(* Logix 5000 project; controller R5_CSS vendor 1 type 14 code 74 rev 19.11; software revision 19.01; part 11 of 18 *)
(* tags used below, declared in another part *)
   P205 : PUMP_CONTROL;   // OVERHEAD CONDENSER TRANSFER PUMP
   PC101 : PRESSURE_CONTROL;   // Upper quench tower Diff Pressure
   PC101A : PRESSURE_CONTROL;   // LOWER QUENCH TOWER PRESSURE TRANSMITTER
   PC101B : PRESSURE_CONTROL;   // UPPER QUENCH TOWER PRESSURE TRANSMITTER PRESSURE CONTOL
   PC102A : PRESSURE_CONTROL;   // QUENCH BASIN TRANSFER PUMP SUCTION PRESSURE CONTROL
   PC102B : PRESSURE_CONTROL;   // QUENCH BASIN TRANSFER PUMP DISCHARGE PRESSURE CONTROL
   PC132 : PRESSURE_CONTROL;
   PC132_AUTO_Ons : BOOL;
   PC132_AUTO_Ons1 : BOOL;
   PC132_PID : PID;
   PC132_PID_TON : TIMER;
   PC133 : PRESSURE_CONTROL;
   PC133_AUTO_Ons : BOOL;
   PC133_AUTO_Ons1 : BOOL;
   PC133_PID : PID;
   PC133_PID_TON : TIMER;
   Test : INT[500];
   TMR_CRIT_FAULT : DINT;
   TMR_FAULT : DINT;
(* MainProgram, continued *)

ROUTINE PC101_QuenchTowerPressureDelta   (* ladder *)
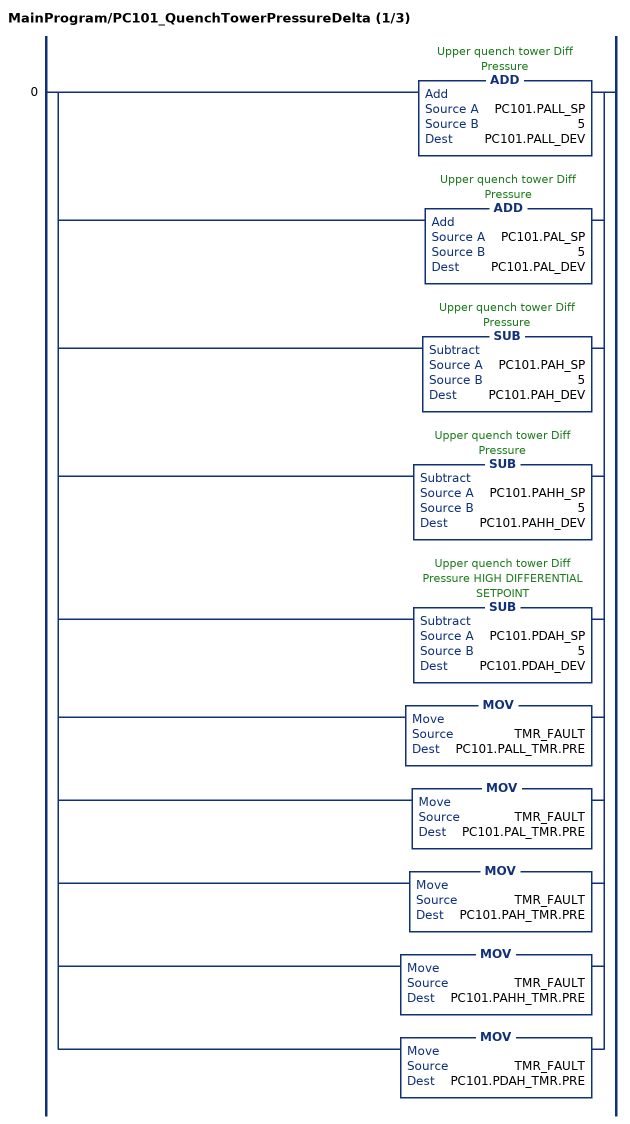
   0: [ADD(PC101.PALL_SP,5,PC101.PALL_DEV) ,ADD(PC101.PAL_SP,5,PC101.PAL_DEV) ,SUB(PC101.PAH_SP,5,PC101.PAH_DEV) ,SUB(PC101.PAHH_SP,5,PC101.PAHH_DEV) ,SUB(PC101.PDAH_SP,5,PC101.PDAH_DEV) ,MOV(TMR_FAULT,PC101.PALL_TMR.PRE) ,MOV(TMR_FAULT,PC101.PAL_TMR.PRE) ,MOV(TMR_FAULT,PC101.PAH_TMR.PRE) ,MOV(TMR_FAULT,PC101.PAHH_TMR.PRE) ,MOV(TMR_FAULT,PC101.PDAH_TMR.PRE) ];
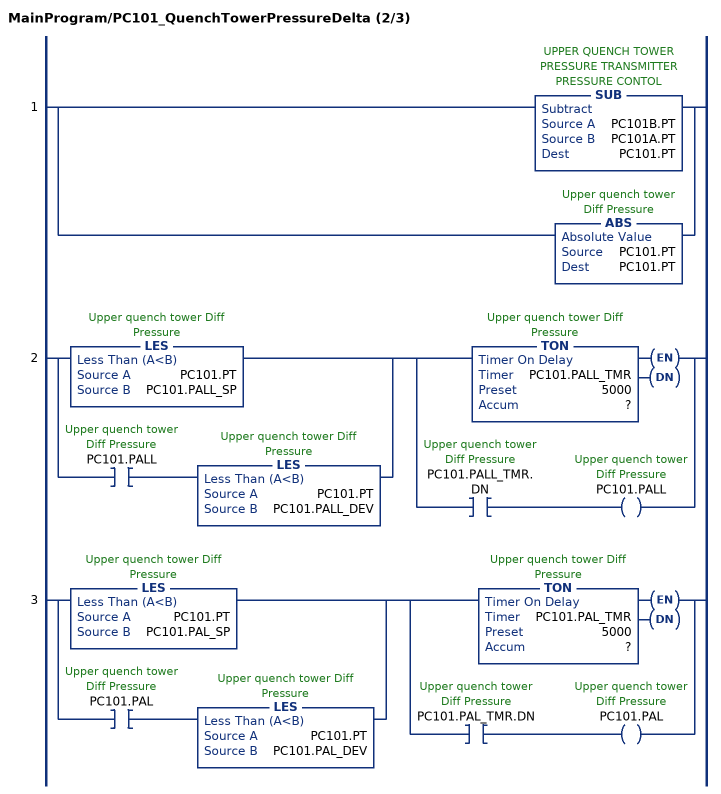
   1: [SUB(PC101B.PT,PC101A.PT,PC101.PT) ,ABS(PC101.PT,PC101.PT) ];
   2: [LES(PC101.PT,PC101.PALL_SP) ,XIC(PC101.PALL) LES(PC101.PT,PC101.PALL_DEV) ][TON(PC101.PALL_TMR,?,?) ,XIC(PC101.PALL_TMR.DN) OTE(PC101.PALL) ];
   3: [LES(PC101.PT,PC101.PAL_SP) ,XIC(PC101.PAL) LES(PC101.PT,PC101.PAL_DEV) ][TON(PC101.PAL_TMR,?,?) ,XIC(PC101.PAL_TMR.DN) OTE(PC101.PAL) ];
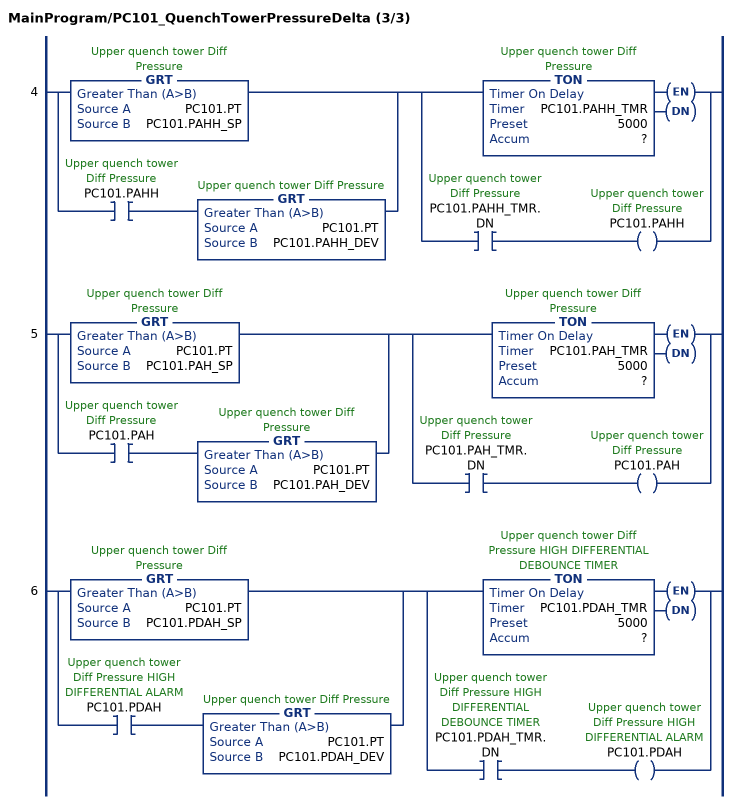
   4: [GRT(PC101.PT,PC101.PAHH_SP) ,XIC(PC101.PAHH) GRT(PC101.PT,PC101.PAHH_DEV) ][TON(PC101.PAHH_TMR,?,?) ,XIC(PC101.PAHH_TMR.DN) OTE(PC101.PAHH) ];
   5: [GRT(PC101.PT,PC101.PAH_SP) ,XIC(PC101.PAH) GRT(PC101.PT,PC101.PAH_DEV) ][TON(PC101.PAH_TMR,?,?) ,XIC(PC101.PAH_TMR.DN) OTE(PC101.PAH) ];
   6: [GRT(PC101.PT,PC101.PDAH_SP) ,XIC(PC101.PDAH) GRT(PC101.PT,PC101.PDAH_DEV) ][TON(PC101.PDAH_TMR,?,?) ,XIC(PC101.PDAH_TMR.DN) OTE(PC101.PDAH) ];
END_ROUTINE

ROUTINE PC101A_QuenchTowerPressure   (* ladder *)
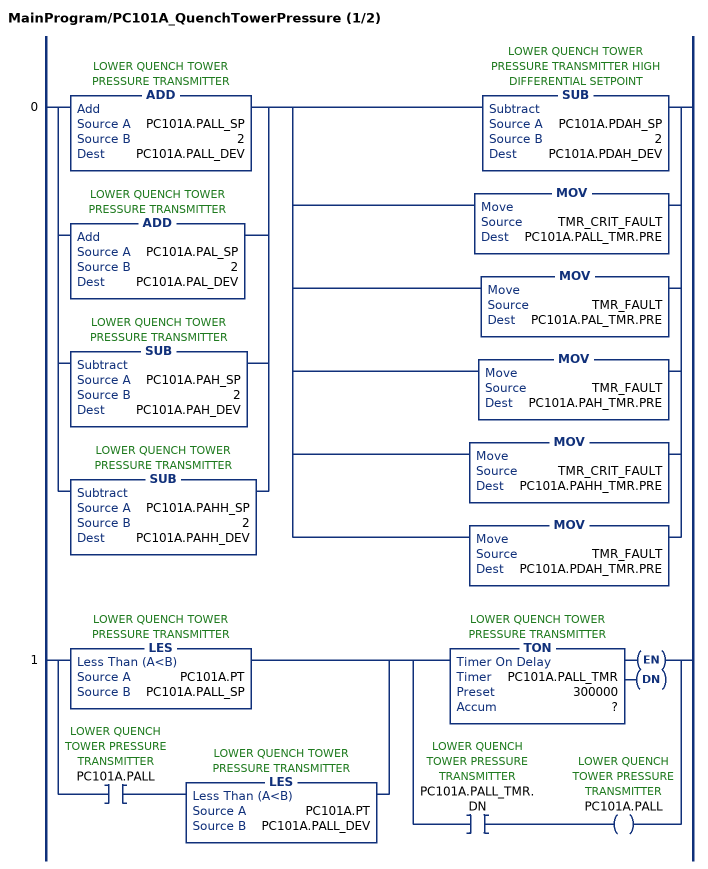
   0: [ADD(PC101A.PALL_SP,2,PC101A.PALL_DEV) ,ADD(PC101A.PAL_SP,2,PC101A.PAL_DEV) ,SUB(PC101A.PAH_SP,2,PC101A.PAH_DEV) ,SUB(PC101A.PAHH_SP,2,PC101A.PAHH_DEV) ][SUB(PC101A.PDAH_SP,2,PC101A.PDAH_DEV) ,MOV(TMR_CRIT_FAULT,PC101A.PALL_TMR.PRE) ,MOV(TMR_FAULT,PC101A.PAL_TMR.PRE) ,MOV(TMR_FAULT,PC101A.PAH_TMR.PRE) ,MOV(TMR_CRIT_FAULT,PC101A.PAHH_TMR.PRE) ,MOV(TMR_FAULT,PC101A.PDAH_TMR.PRE) ];
   1: [LES(PC101A.PT,PC101A.PALL_SP) ,XIC(PC101A.PALL) LES(PC101A.PT,PC101A.PALL_DEV) ][TON(PC101A.PALL_TMR,?,?) ,XIC(PC101A.PALL_TMR.DN) OTE(PC101A.PALL) ];
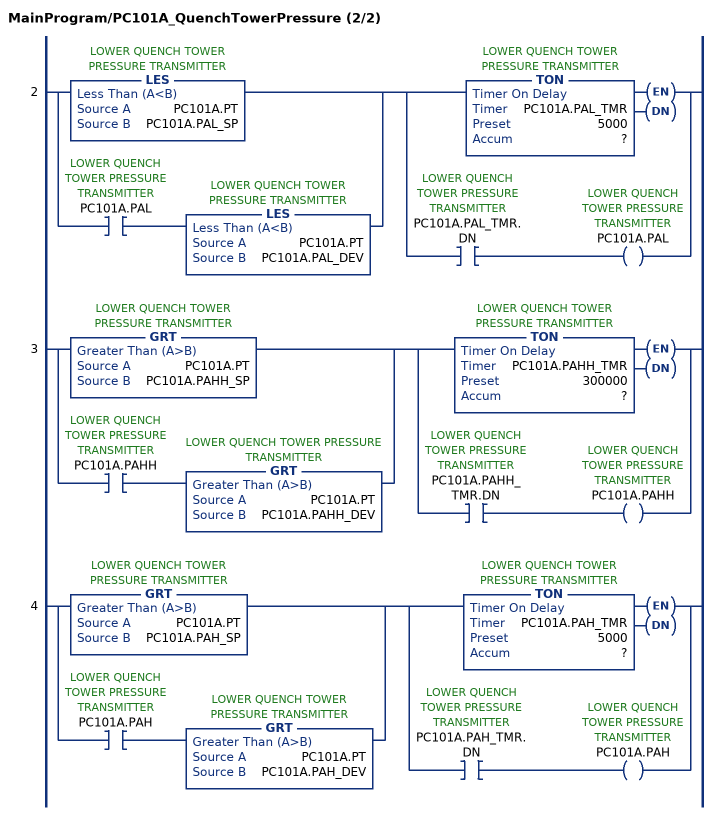
   2: [LES(PC101A.PT,PC101A.PAL_SP) ,XIC(PC101A.PAL) LES(PC101A.PT,PC101A.PAL_DEV) ][TON(PC101A.PAL_TMR,?,?) ,XIC(PC101A.PAL_TMR.DN) OTE(PC101A.PAL) ];
   3: [GRT(PC101A.PT,PC101A.PAHH_SP) ,XIC(PC101A.PAHH) GRT(PC101A.PT,PC101A.PAHH_DEV) ][TON(PC101A.PAHH_TMR,?,?) ,XIC(PC101A.PAHH_TMR.DN) OTE(PC101A.PAHH) ];
   4: [GRT(PC101A.PT,PC101A.PAH_SP) ,XIC(PC101A.PAH) GRT(PC101A.PT,PC101A.PAH_DEV) ][TON(PC101A.PAH_TMR,?,?) ,XIC(PC101A.PAH_TMR.DN) OTE(PC101A.PAH) ];
END_ROUTINE

ROUTINE PC101B_QuenchTowerPressure   (* ladder *)
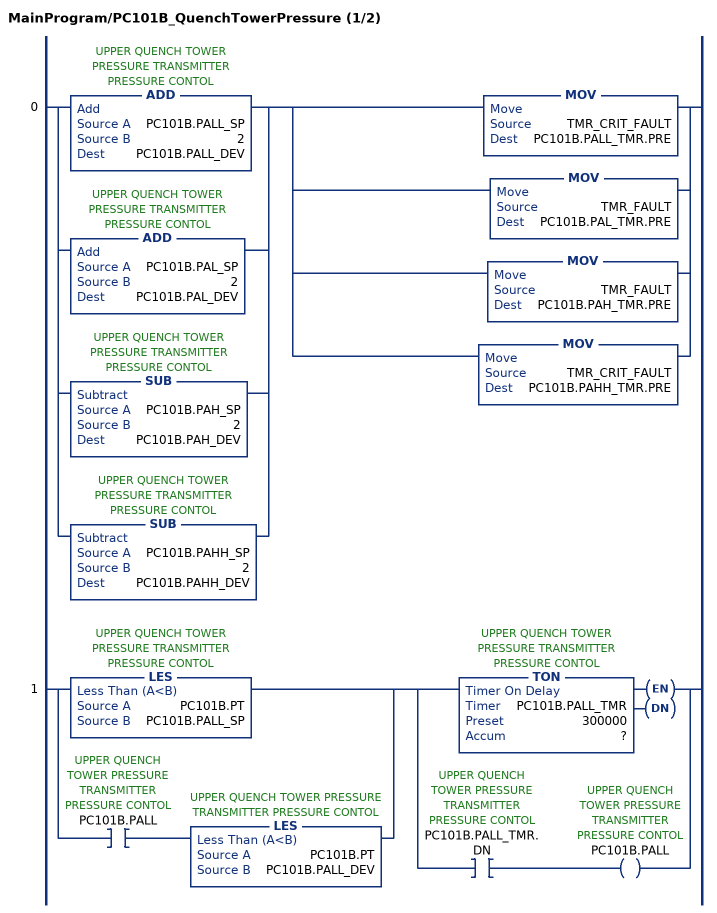
   0: [ADD(PC101B.PALL_SP,2,PC101B.PALL_DEV) ,ADD(PC101B.PAL_SP,2,PC101B.PAL_DEV) ,SUB(PC101B.PAH_SP,2,PC101B.PAH_DEV) ,SUB(PC101B.PAHH_SP,2,PC101B.PAHH_DEV) ][MOV(TMR_CRIT_FAULT,PC101B.PALL_TMR.PRE) ,MOV(TMR_FAULT,PC101B.PAL_TMR.PRE) ,MOV(TMR_FAULT,PC101B.PAH_TMR.PRE) ,MOV(TMR_CRIT_FAULT,PC101B.PAHH_TMR.PRE) ];
   1: [LES(PC101B.PT,PC101B.PALL_SP) ,XIC(PC101B.PALL) LES(PC101B.PT,PC101B.PALL_DEV) ][TON(PC101B.PALL_TMR,?,?) ,XIC(PC101B.PALL_TMR.DN) OTE(PC101B.PALL) ];
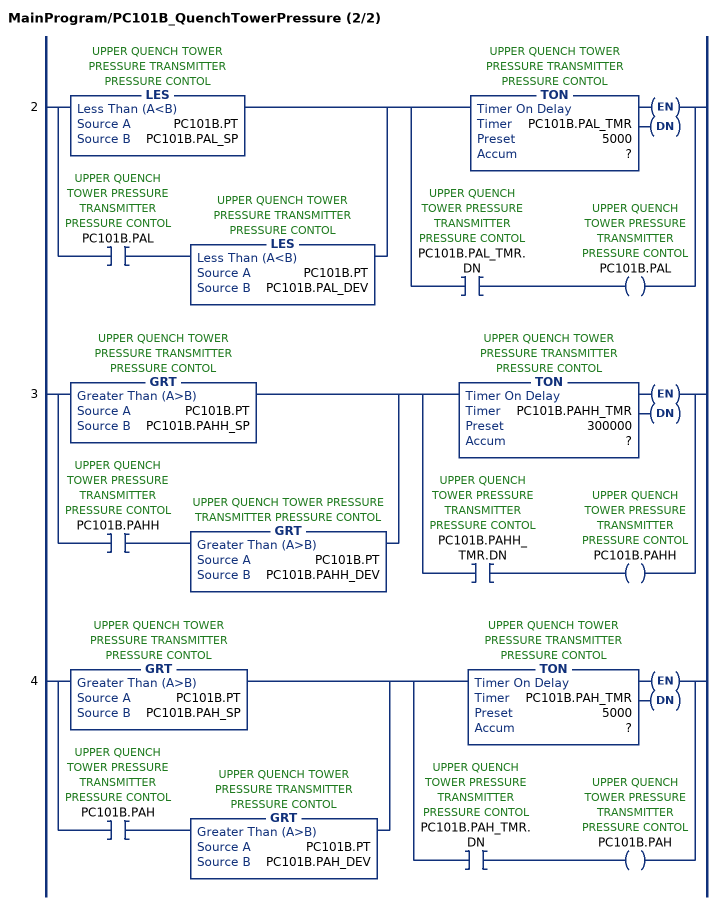
   2: [LES(PC101B.PT,PC101B.PAL_SP) ,XIC(PC101B.PAL) LES(PC101B.PT,PC101B.PAL_DEV) ][TON(PC101B.PAL_TMR,?,?) ,XIC(PC101B.PAL_TMR.DN) OTE(PC101B.PAL) ];
   3: [GRT(PC101B.PT,PC101B.PAHH_SP) ,XIC(PC101B.PAHH) GRT(PC101B.PT,PC101B.PAHH_DEV) ][TON(PC101B.PAHH_TMR,?,?) ,XIC(PC101B.PAHH_TMR.DN) OTE(PC101B.PAHH) ];
   4: [GRT(PC101B.PT,PC101B.PAH_SP) ,XIC(PC101B.PAH) GRT(PC101B.PT,PC101B.PAH_DEV) ][TON(PC101B.PAH_TMR,?,?) ,XIC(PC101B.PAH_TMR.DN) OTE(PC101B.PAH) ];
END_ROUTINE

ROUTINE PC102A_PumpSuctionHead   (* ladder *)
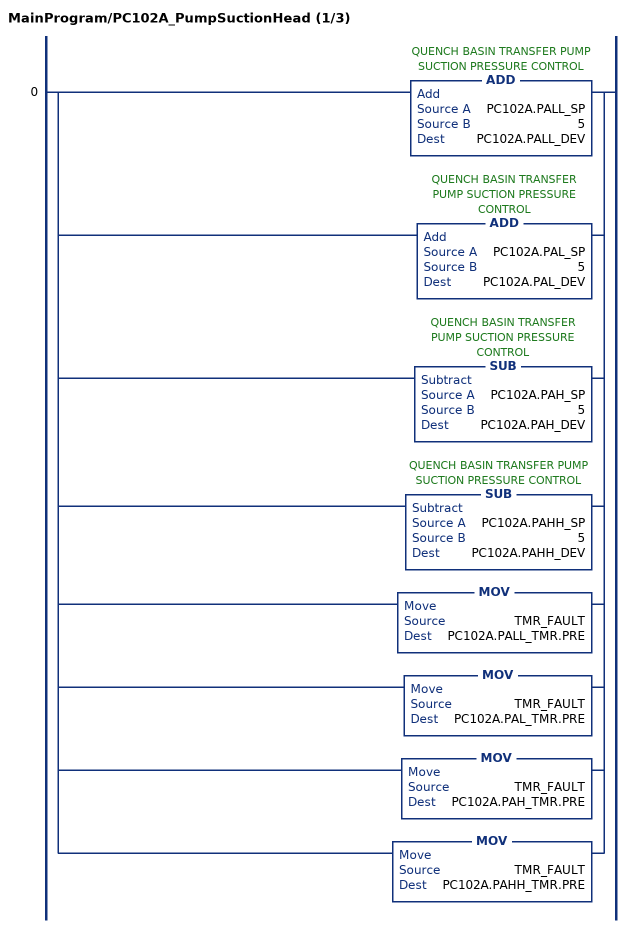
   0: [ADD(PC102A.PALL_SP,5,PC102A.PALL_DEV) ,ADD(PC102A.PAL_SP,5,PC102A.PAL_DEV) ,SUB(PC102A.PAH_SP,5,PC102A.PAH_DEV) ,SUB(PC102A.PAHH_SP,5,PC102A.PAHH_DEV) ,MOV(TMR_FAULT,PC102A.PALL_TMR.PRE) ,MOV(TMR_FAULT,PC102A.PAL_TMR.PRE) ,MOV(TMR_FAULT,PC102A.PAH_TMR.PRE) ,MOV(TMR_FAULT,PC102A.PAHH_TMR.PRE) ];
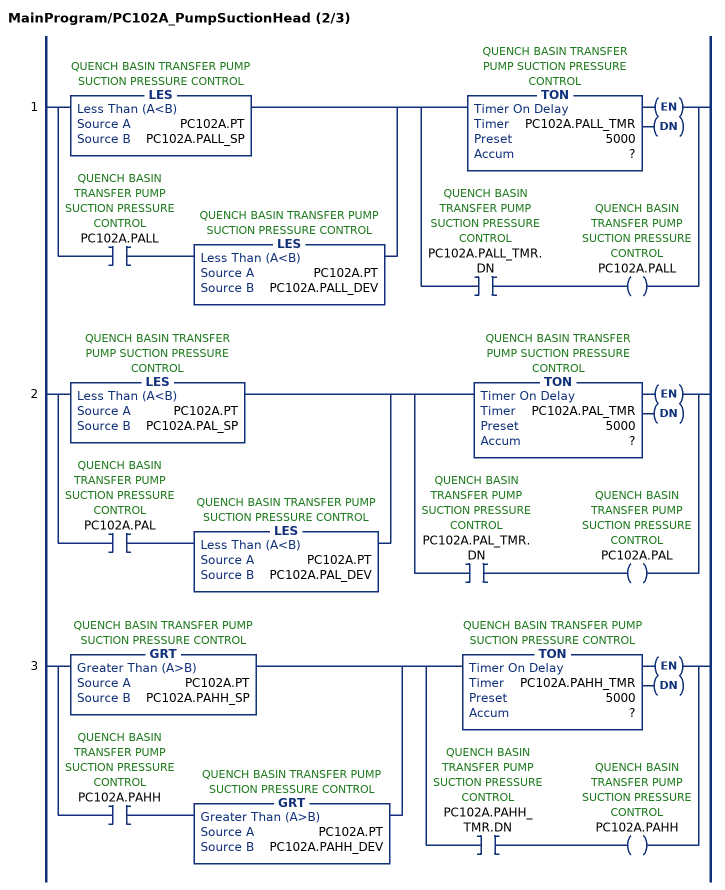
   1: [LES(PC102A.PT,PC102A.PALL_SP) ,XIC(PC102A.PALL) LES(PC102A.PT,PC102A.PALL_DEV) ][TON(PC102A.PALL_TMR,?,?) ,XIC(PC102A.PALL_TMR.DN) OTE(PC102A.PALL) ];
   2: [LES(PC102A.PT,PC102A.PAL_SP) ,XIC(PC102A.PAL) LES(PC102A.PT,PC102A.PAL_DEV) ][TON(PC102A.PAL_TMR,?,?) ,XIC(PC102A.PAL_TMR.DN) OTE(PC102A.PAL) ];
   3: [GRT(PC102A.PT,PC102A.PAHH_SP) ,XIC(PC102A.PAHH) GRT(PC102A.PT,PC102A.PAHH_DEV) ][TON(PC102A.PAHH_TMR,?,?) ,XIC(PC102A.PAHH_TMR.DN) OTE(PC102A.PAHH) ];
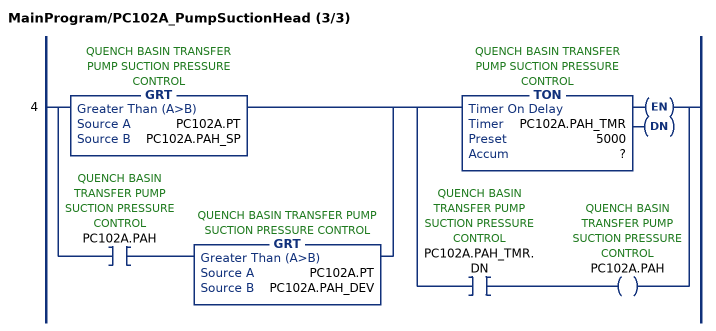
   4: [GRT(PC102A.PT,PC102A.PAH_SP) ,XIC(PC102A.PAH) GRT(PC102A.PT,PC102A.PAH_DEV) ][TON(PC102A.PAH_TMR,?,?) ,XIC(PC102A.PAH_TMR.DN) OTE(PC102A.PAH) ];
END_ROUTINE

ROUTINE PC102B_BasinPumpDischargePress   (* ladder *)
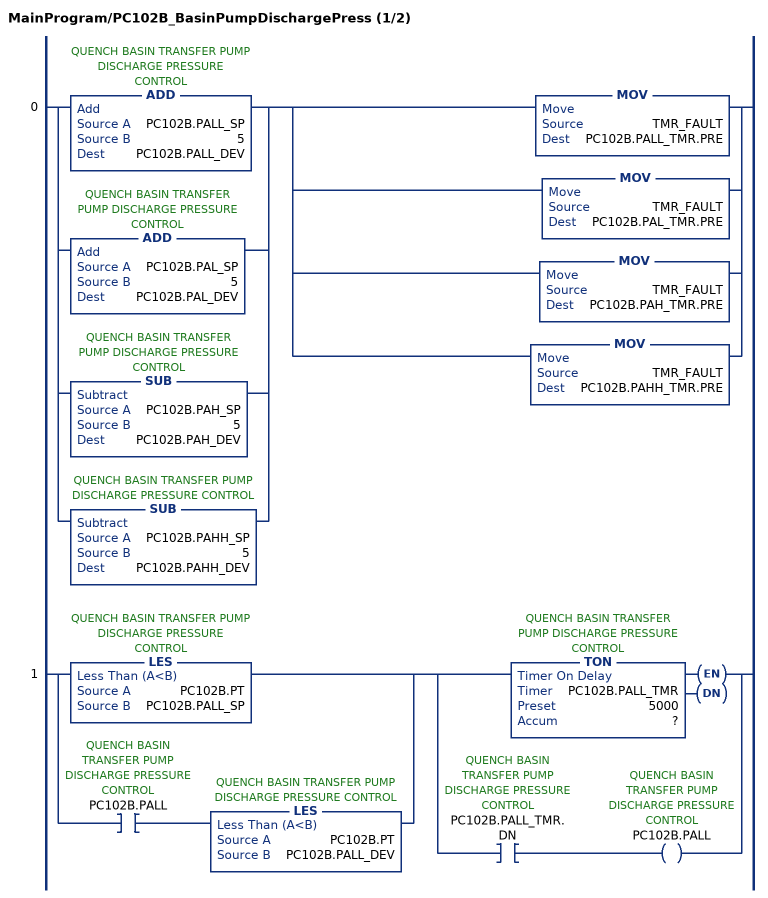
   0: [ADD(PC102B.PALL_SP,5,PC102B.PALL_DEV) ,ADD(PC102B.PAL_SP,5,PC102B.PAL_DEV) ,SUB(PC102B.PAH_SP,5,PC102B.PAH_DEV) ,SUB(PC102B.PAHH_SP,5,PC102B.PAHH_DEV) ][MOV(TMR_FAULT,PC102B.PALL_TMR.PRE) ,MOV(TMR_FAULT,PC102B.PAL_TMR.PRE) ,MOV(TMR_FAULT,PC102B.PAH_TMR.PRE) ,MOV(TMR_FAULT,PC102B.PAHH_TMR.PRE) ];
   1: [LES(PC102B.PT,PC102B.PALL_SP) ,XIC(PC102B.PALL) LES(PC102B.PT,PC102B.PALL_DEV) ][TON(PC102B.PALL_TMR,?,?) ,XIC(PC102B.PALL_TMR.DN) OTE(PC102B.PALL) ];
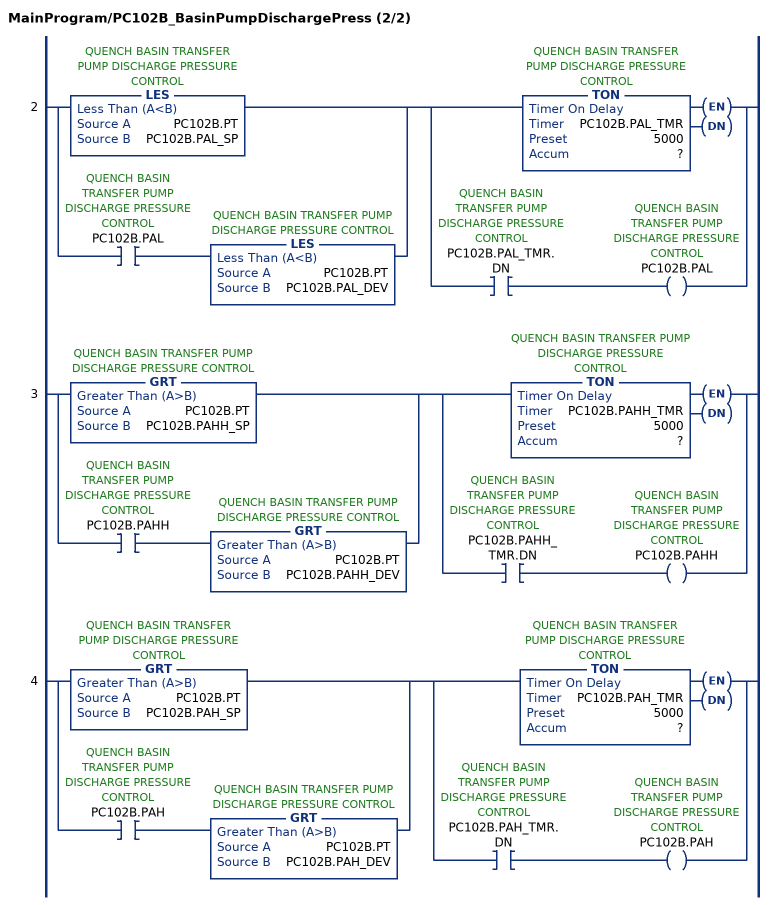
   2: [LES(PC102B.PT,PC102B.PAL_SP) ,XIC(PC102B.PAL) LES(PC102B.PT,PC102B.PAL_DEV) ][TON(PC102B.PAL_TMR,?,?) ,XIC(PC102B.PAL_TMR.DN) OTE(PC102B.PAL) ];
   3: [GRT(PC102B.PT,PC102B.PAHH_SP) ,XIC(PC102B.PAHH) GRT(PC102B.PT,PC102B.PAHH_DEV) ][TON(PC102B.PAHH_TMR,?,?) ,XIC(PC102B.PAHH_TMR.DN) OTE(PC102B.PAHH) ];
   4: [GRT(PC102B.PT,PC102B.PAH_SP) ,XIC(PC102B.PAH) GRT(PC102B.PT,PC102B.PAH_DEV) ][TON(PC102B.PAH_TMR,?,?) ,XIC(PC102B.PAH_TMR.DN) OTE(PC102B.PAH) ];
END_ROUTINE

ROUTINE PC132_GTL1_Pressure_PID   (* ladder *)
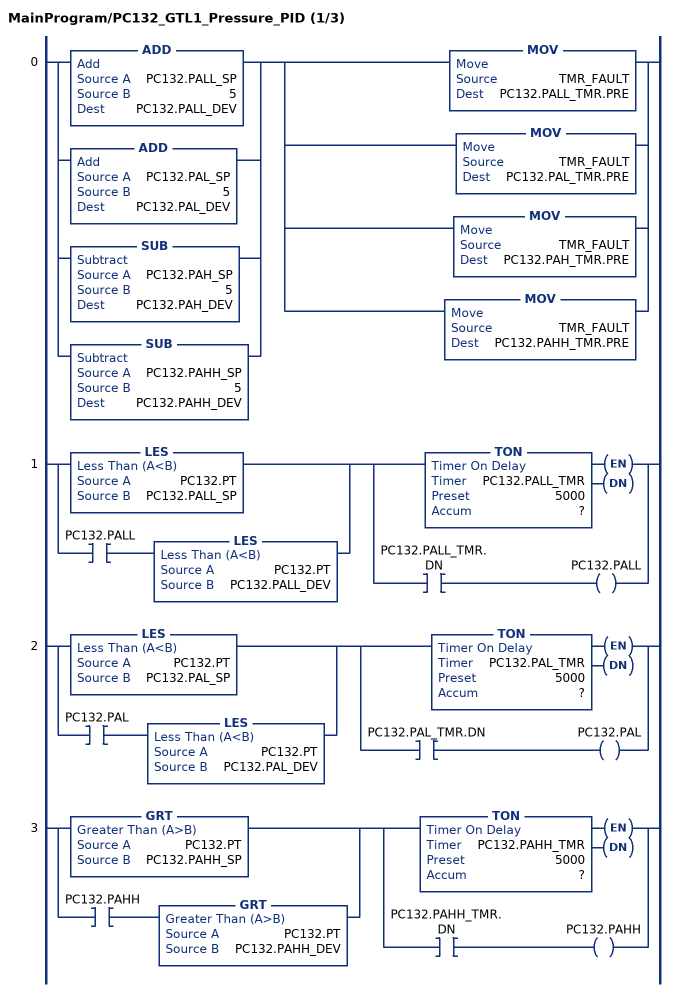
   0: [ADD(PC132.PALL_SP,5,PC132.PALL_DEV) ,ADD(PC132.PAL_SP,5,PC132.PAL_DEV) ,SUB(PC132.PAH_SP,5,PC132.PAH_DEV) ,SUB(PC132.PAHH_SP,5,PC132.PAHH_DEV) ][MOV(TMR_FAULT,PC132.PALL_TMR.PRE) ,MOV(TMR_FAULT,PC132.PAL_TMR.PRE) ,MOV(TMR_FAULT,PC132.PAH_TMR.PRE) ,MOV(TMR_FAULT,PC132.PAHH_TMR.PRE) ];
   1: [LES(PC132.PT,PC132.PALL_SP) ,XIC(PC132.PALL) LES(PC132.PT,PC132.PALL_DEV) ][TON(PC132.PALL_TMR,?,?) ,XIC(PC132.PALL_TMR.DN) OTE(PC132.PALL) ];
   2: [LES(PC132.PT,PC132.PAL_SP) ,XIC(PC132.PAL) LES(PC132.PT,PC132.PAL_DEV) ][TON(PC132.PAL_TMR,?,?) ,XIC(PC132.PAL_TMR.DN) OTE(PC132.PAL) ];
   3: [GRT(PC132.PT,PC132.PAHH_SP) ,XIC(PC132.PAHH) GRT(PC132.PT,PC132.PAHH_DEV) ][TON(PC132.PAHH_TMR,?,?) ,XIC(PC132.PAHH_TMR.DN) OTE(PC132.PAHH) ];
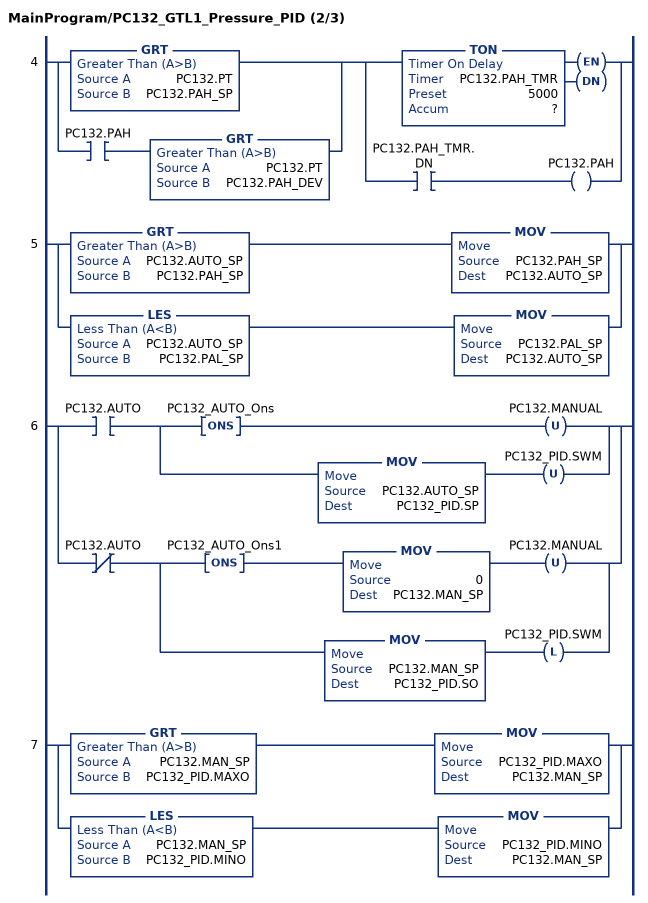
   4: [GRT(PC132.PT,PC132.PAH_SP) ,XIC(PC132.PAH) GRT(PC132.PT,PC132.PAH_DEV) ][TON(PC132.PAH_TMR,?,?) ,XIC(PC132.PAH_TMR.DN) OTE(PC132.PAH) ];
   5: [GRT(PC132.AUTO_SP,PC132.PAH_SP) MOV(PC132.PAH_SP,PC132.AUTO_SP) ,LES(PC132.AUTO_SP,PC132.PAL_SP) MOV(PC132.PAL_SP,PC132.AUTO_SP) ];
   6: [XIC(PC132.AUTO) [ONS(PC132_AUTO_Ons) OTU(PC132.MANUAL) ,MOV(PC132.AUTO_SP,PC132_PID.SP) OTU(PC132_PID.SWM) ] ,XIO(PC132.AUTO) [ONS(PC132_AUTO_Ons1) MOV(0,PC132.MAN_SP) OTU(PC132.MANUAL) ,MOV(PC132.MAN_SP,PC132_PID.SO) OTL(PC132_PID.SWM) ] ];
   7: [GRT(PC132.MAN_SP,PC132_PID.MAXO) MOV(PC132_PID.MAXO,PC132.MAN_SP) ,LES(PC132.MAN_SP,PC132_PID.MINO) MOV(PC132_PID.MINO,PC132.MAN_SP) ];
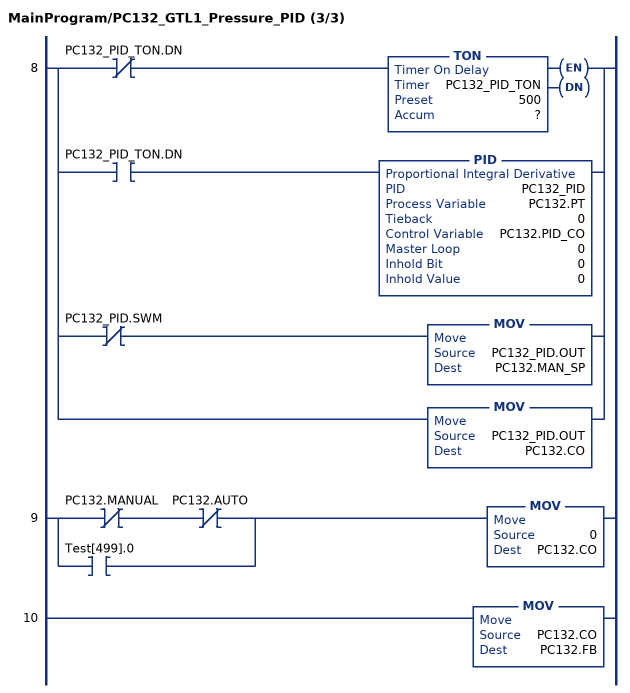
   8: [XIO(PC132_PID_TON.DN) TON(PC132_PID_TON,?,?) ,XIC(PC132_PID_TON.DN) PID(PC132_PID,PC132.PT,0,PC132.PID_CO,0,0,0) ,XIO(PC132_PID.SWM) MOV(PC132_PID.OUT,PC132.MAN_SP) ,MOV(PC132_PID.OUT,PC132.CO) ];
   9: [XIO(PC132.MANUAL) XIO(PC132.AUTO) ,XIC(Test[499].0) ]MOV(0,PC132.CO);
   10: MOV(PC132.CO,PC132.FB);
END_ROUTINE

ROUTINE PC133_GTL2_Pressure_PID   (* ladder *)
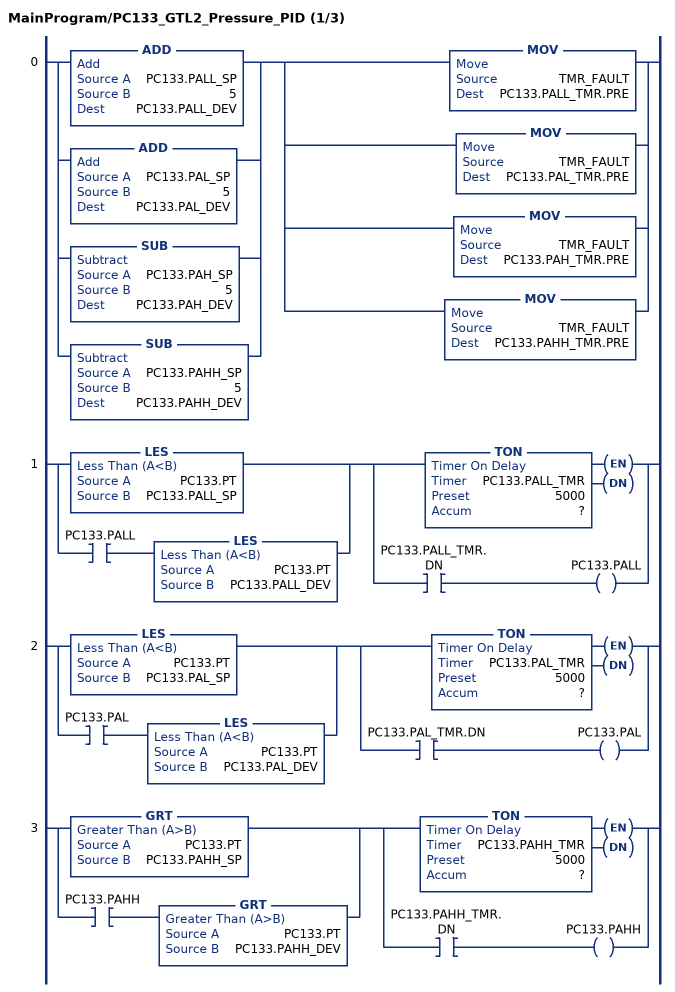
   0: [ADD(PC133.PALL_SP,5,PC133.PALL_DEV) ,ADD(PC133.PAL_SP,5,PC133.PAL_DEV) ,SUB(PC133.PAH_SP,5,PC133.PAH_DEV) ,SUB(PC133.PAHH_SP,5,PC133.PAHH_DEV) ][MOV(TMR_FAULT,PC133.PALL_TMR.PRE) ,MOV(TMR_FAULT,PC133.PAL_TMR.PRE) ,MOV(TMR_FAULT,PC133.PAH_TMR.PRE) ,MOV(TMR_FAULT,PC133.PAHH_TMR.PRE) ];
   1: [LES(PC133.PT,PC133.PALL_SP) ,XIC(PC133.PALL) LES(PC133.PT,PC133.PALL_DEV) ][TON(PC133.PALL_TMR,?,?) ,XIC(PC133.PALL_TMR.DN) OTE(PC133.PALL) ];
   2: [LES(PC133.PT,PC133.PAL_SP) ,XIC(PC133.PAL) LES(PC133.PT,PC133.PAL_DEV) ][TON(PC133.PAL_TMR,?,?) ,XIC(PC133.PAL_TMR.DN) OTE(PC133.PAL) ];
   3: [GRT(PC133.PT,PC133.PAHH_SP) ,XIC(PC133.PAHH) GRT(PC133.PT,PC133.PAHH_DEV) ][TON(PC133.PAHH_TMR,?,?) ,XIC(PC133.PAHH_TMR.DN) OTE(PC133.PAHH) ];
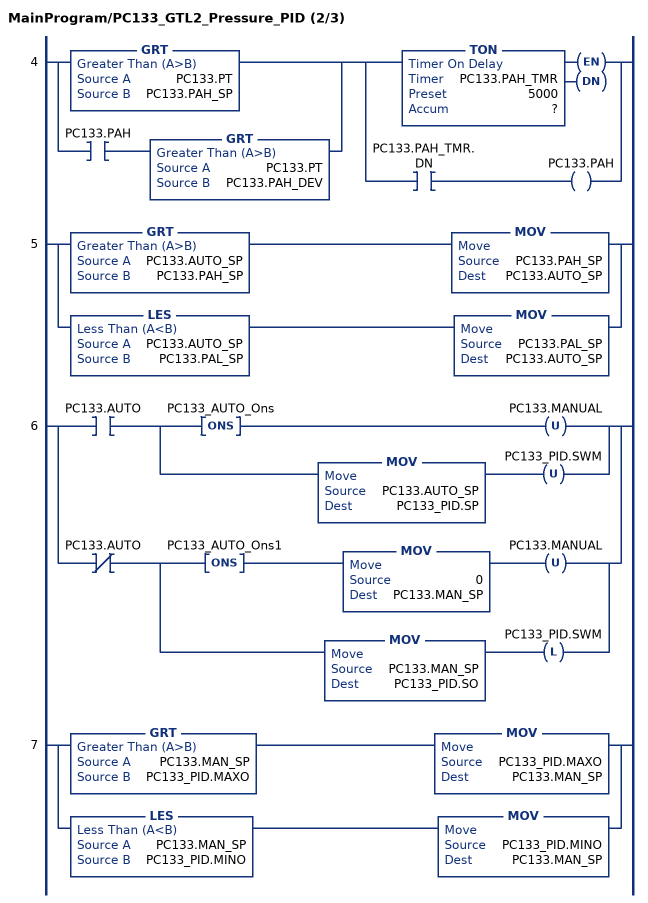
   4: [GRT(PC133.PT,PC133.PAH_SP) ,XIC(PC133.PAH) GRT(PC133.PT,PC133.PAH_DEV) ][TON(PC133.PAH_TMR,?,?) ,XIC(PC133.PAH_TMR.DN) OTE(PC133.PAH) ];
   5: [GRT(PC133.AUTO_SP,PC133.PAH_SP) MOV(PC133.PAH_SP,PC133.AUTO_SP) ,LES(PC133.AUTO_SP,PC133.PAL_SP) MOV(PC133.PAL_SP,PC133.AUTO_SP) ];
   6: [XIC(PC133.AUTO) [ONS(PC133_AUTO_Ons) OTU(PC133.MANUAL) ,MOV(PC133.AUTO_SP,PC133_PID.SP) OTU(PC133_PID.SWM) ] ,XIO(PC133.AUTO) [ONS(PC133_AUTO_Ons1) MOV(0,PC133.MAN_SP) OTU(PC133.MANUAL) ,MOV(PC133.MAN_SP,PC133_PID.SO) OTL(PC133_PID.SWM) ] ];
   7: [GRT(PC133.MAN_SP,PC133_PID.MAXO) MOV(PC133_PID.MAXO,PC133.MAN_SP) ,LES(PC133.MAN_SP,PC133_PID.MINO) MOV(PC133_PID.MINO,PC133.MAN_SP) ];
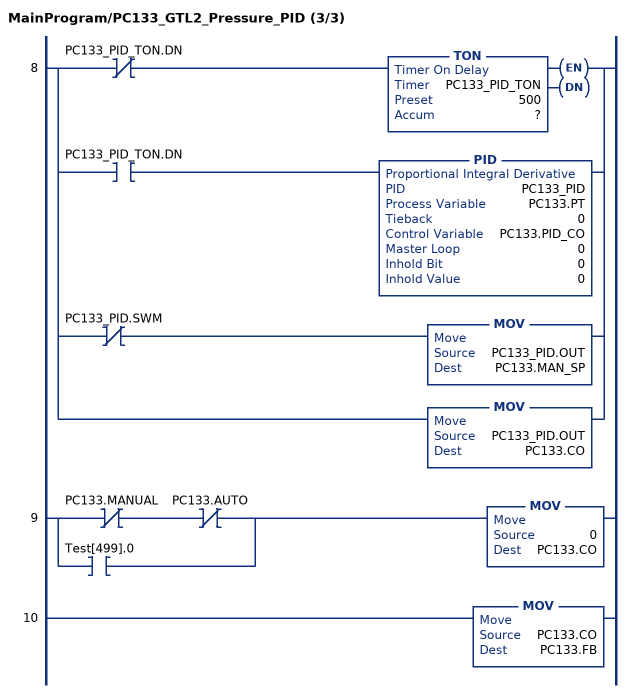
   8: [XIO(PC133_PID_TON.DN) TON(PC133_PID_TON,?,?) ,XIC(PC133_PID_TON.DN) PID(PC133_PID,PC133.PT,0,PC133.PID_CO,0,0,0) ,XIO(PC133_PID.SWM) MOV(PC133_PID.OUT,PC133.MAN_SP) ,MOV(PC133_PID.OUT,PC133.CO) ];
   9: [XIO(PC133.MANUAL) XIO(PC133.AUTO) ,XIC(Test[499].0) ]MOV(0,PC133.CO);
   10: MOV(PC133.CO,PC133.FB);
END_ROUTINE
